(* IEC 61131-3 sources: moqui-plc/iec61131/moqui/framework/src/main/org/moqui/mqtt, 14 files *)

(* ---- MqttCmd.dut ---- *)
(*#-#-#-#-#-#-#-#-#-#---Declaration---#-#-#-#-#-#-#-#-#-#-#-#-#*)

{attribute 'qualified_only'}
{attribute 'strict'}
TYPE MqttCmd : (
	Idle := 0,
	Publish,
    Subscribe,
	Unsubscribe
); END_TYPE

(* ---- MqttCmd.st ---- *)
TYPE MqttCmd : (
	Idle := 0,
	Publish,
    Subscribe,
	Unsubscribe
); END_TYPE

(* ---- MqttConnectionRef.dut ---- *)
(*#-#-#-#-#-#-#-#-#-#---Declaration---#-#-#-#-#-#-#-#-#-#-#-#-#*)

TYPE MqttConnectionRef : STRUCT
	ref : REFERENCE TO MQTT.MQTTClient;
END_STRUCT END_TYPE

(* ---- MqttConnectionRef.st ---- *)
TYPE MqttConnectionRef : STRUCT
	ref : REFERENCE TO MQTT.MQTTClient;
END_STRUCT END_TYPE

(* ---- MqttLogAppenderStatus.dut ---- *)
(*#-#-#-#-#-#-#-#-#-#---Declaration---#-#-#-#-#-#-#-#-#-#-#-#-#*)

{attribute 'qualified_only'}
{attribute 'strict'}
TYPE MqttLogAppenderStatus : (
    Idle,
	BuildJson,
	Serialize,
	Publish,
	WaitAck
); END_TYPE

(* ---- MqttLogAppenderStatus.st ---- *)
TYPE MqttLogAppenderStatus : (
    Idle,
	BuildJson,
	Serialize,
	Publish,
	WaitAck
); END_TYPE

(* ---- MqttParameterPubStatus.dut ---- *)
(*#-#-#-#-#-#-#-#-#-#---Declaration---#-#-#-#-#-#-#-#-#-#-#-#-#*)

{attribute 'qualified_only'}
{attribute 'strict'}
TYPE MqttParameterPubStatus : (
	Idle := 0,
	BuildJson,
	Serialize,
	Publish,
	WaitAck
); END_TYPE

(* ---- MqttParameterPubStatus.st ---- *)
TYPE MqttParameterPubStatus : (
	Idle := 0,
	BuildJson,
	Serialize,
	Publish,
	WaitAck
); END_TYPE

(* ---- MqttParameterSubStatus.dut ---- *)
(*#-#-#-#-#-#-#-#-#-#---Declaration---#-#-#-#-#-#-#-#-#-#-#-#-#*)

{attribute 'qualified_only'}
{attribute 'strict'}
TYPE MqttParameterSubStatus : (
	Idle := 0,
	Subscribe,
	UpdateParameters,
	Listening,
	Error
); END_TYPE

(* ---- MqttParameterSubStatus.st ---- *)
TYPE MqttParameterSubStatus : (
	Idle := 0,
	Subscribe,
	UpdateParameters,
	Listening,
	Error
); END_TYPE

(* ---- MqttConnectionFactory.pou ---- *)
(*#-#-#-#-#-#-#-#-#-#---Declaration---#-#-#-#-#-#-#-#-#-#-#-#-#*)

{attribute 'no_assign'}
(* Component to connect with a MQTT broker, using default configurations. *)
FUNCTION_BLOCK MqttConnectionFactory
VAR_EXTERNAL CONSTANT
	brokerUrl : STRING(255);
	brokerPort : UINT;
	webSocketUrl : STRING(1024);
	clientId : STRING(255);
	username : WSTRING(255);
	password : WSTRING(1024);
	sessionExpiryInterval : UDINT;
	keepAlive : UINT;
	cleanSession : BOOL;
	timeout : UDINT;
	pingInterval : TIME;
	maximumPacketSize : UDINT;
	communicationMode : MQTT.COMMUNICATION_MODE;
	mqttVersion : MQTT.MQTT_VERSION;
	(* connectUserProperties : ARRAY [0..(MQTT.MQTTParam.g_udiMaxUserProperties - 1)] OF MQTT.MQTTStringPair; *)
	willTopic : WSTRING(1024);
	willMessage : STRING(1024);
	willRetain : BOOL;
	willQoS : MQTT.MQTT_QOS;
	willPayloadFormatIndicator : BYTE;
	willMessageExpiryInterval : UDINT;
	willContentType : WSTRING(32);
	willDelayInterval : UDINT;
END_VAR
VAR_INPUT
	connect : BOOL := TRUE;
END_VAR
VAR_OUTPUT
	connection : MQTT.MQTTClient;
    connected : BOOL;
    busy : BOOL;
    error : BOOL;
	errorId : INT;
END_VAR
VAR
	(* Connect properties v5 *)
	mqttConnectProperties : MQTT.MQTTConnectProperties := (
		udiSessionExpiryInterval := sessionExpiryInterval,
		udiMaximumPacketSize := maximumPacketSize
		(* userProperties := connectUserProperties *)
	);
	(* Will properties v5 *)
	mqttWillProperties : MQTT.MQTTWillProperties := (
		bPayloadFormatIndicator := willPayloadFormatIndicator,
		udiMessageExpiryInterval := willMessageExpiryInterval,
		wsContentType := willContentType,
		udiWillDelayInterval := willDelayInterval
		(* userProperties := willUserProperties *)
    );
	(* TLS context *)
	cipherList : NBS.CIPHER_LIST := STRUCT(psList := ADR('HIGH'), udiSize := 5);
	commonName : STRING := 'moqui';
    certInfo : NBS.CERT_INFO := (psInfo := ADR(commonName), udiSize := INT_TO_UDINT(LEN(commonName)));
	defaultTlsContext : NBS.TLSContext := (
		sUseCaseName := commonName,
		ePurpose := NBS.PURPOSE.CLIENT_SIDE,
		sTLSVersion := '1.3',
		sCipherList := cipherList,
		sHostname := brokerUrl,
		ciCertInfo := certInfo,
		udiVerificationMode	:= 2, (* 1 => No peer verification, 2 => Active Peer verification *)
		itfCertVerifer := 0
	);
	nullTlsContext : NBS.ITLSContext := 0;
	tlsContext : NBS.ITLSContext;
	useTLS : BOOL := FALSE;

	(*
     * To use client certificates, configure the connection via the TLS context.
	 * Example:
	 *      commonName : STRING := 'COMMON_NAME_OF_CERTIFICATE'; // CN of the certificate (common name).
	 *      cipherList : NBS.CIPHER_LIST := STRUCT(psList := ADR('HIGH'), udiSize := 5); // Cipher string see https://www.openssl.org/docs/man1.1.1/man1/ciphers.html
	 *      certInfo : NBS.CERT_INFO := (psInfo := ADR(commonName), udiSize := SIZEOF(commonName)); // CN of the certificate (common name)
	 *      tlsContext : NBS.TLSContext := (
	 *          sUseCaseName := commonName, // A certificate is stored in the certificate store with the use case name.
	 *          ePurpose := NBS.PURPOSE.CLIENT_SIDE, // For client certificates set this to NBS.PURPOSE.CLIENT_SIDE
     *          sTLSVersion := '1.3', // The TLS version
     *          sCipherList := cipherList, // Set the cipher list
     *          sHostname := brokerUrl, // The hostname of the broker
     *          udiVerificationMode := 2, // 2 => Active Peer verification
     *          ciCertInfo := certInfo, // Set the cert info
     *          itfCertVerifer := 0); // 0 => No Verifier
	 *      client : MQTT.MQTTClient := (itfTLSCOntext := _tlsContext);
	 * Use the method TLSContext.SetInitialValue to set the context while runtime and set the context via the input itfTLSCOntext of the client FB.
	 *)
END_VAR

(*#-#-#-#-#-#-#-#-#-#---Implementation---#-#-#-#-#-#-#-#-#-#-#-#-#*)

(* TLS selection *)
tlsContext := nullTlsContext;
IF useTLS THEN tlsContext := defaultTlsContext; END_IF;

(* Configure the MQTT connection *)
connection(xEnable := connect, xConnectedToBroker => connected, xError => error, eMQTTerror => errorId,
	sHostname := brokerUrl, uiPort := brokerPort, sWebSocketUrl := webSocketUrl, sClientId := clientId,
	itfTLSContext := tlsContext, eCommunicationMode := communicationMode, eMQTTVersion := mqttVersion,
	wsUsername := username, wsPassword := password, mQTTConnectProperties := mqttConnectProperties,
	uiKeepAlive := keepAlive, xCleanSession := cleanSession, udiTimeOut := timeout, tPingInterval := pingInterval,
	wsWillTopic := willTopic, pbWillMessage := ADR(willMessage), uiWillMessageSize := INT_TO_UINT(LEN(willMessage)),
	xWillRetain := willRetain, eWillQoS := willQoS, mQTTWillProperties := mqttWillProperties);

(* ---- MqttConnectionFactory.st ---- *)
(* Component to connect with a MQTT broker, using default configurations. *)
FUNCTION_BLOCK MqttConnectionFactory
	VAR_EXTERNAL CONSTANT
		brokerUrl : STRING(255);
		brokerPort : UINT;
		webSocketUrl : STRING(1024);
		clientId : STRING(255);
		username : WSTRING(255);
		password : WSTRING(1024);
		sessionExpiryInterval : UDINT;
		keepAlive : UINT;
		cleanSession : BOOL;
		timeout : UDINT;
		pingInterval : TIME;
		maximumPacketSize : UDINT;
		communicationMode : MQTT.COMMUNICATION_MODE;
		mqttVersion : MQTT.MQTT_VERSION;
		(* connectUserProperties : ARRAY [0..(MQTT.MQTTParam.g_udiMaxUserProperties - 1)] OF MQTT.MQTTStringPair; *)
		willTopic : WSTRING(1024);
		willMessage : STRING(1024);
		willRetain : BOOL;
		willQoS : MQTT.MQTT_QOS;
		willPayloadFormatIndicator : BYTE;
		willMessageExpiryInterval : UDINT;
		willContentType : WSTRING(32);
		willDelayInterval : UDINT;
	END_VAR
	VAR_INPUT
		connect : BOOL := TRUE;
	END_VAR
	VAR_OUTPUT
		connection : MQTT.MQTTClient;
	    connected : BOOL;
	    busy : BOOL;
	    error : BOOL;
		errorId : INT;
	END_VAR
	VAR
		(* Connect properties v5 *)
		mqttConnectProperties : MQTT.MQTTConnectProperties := (
			udiSessionExpiryInterval := sessionExpiryInterval,
			udiMaximumPacketSize := maximumPacketSize
			(* userProperties := connectUserProperties *)
		);
		(* Will properties v5 *)
		mqttWillProperties : MQTT.MQTTWillProperties := (
			bPayloadFormatIndicator := willPayloadFormatIndicator,
			udiMessageExpiryInterval := willMessageExpiryInterval,
			wsContentType := willContentType,
			udiWillDelayInterval := willDelayInterval
			(* userProperties := willUserProperties *)
	    );
		(* TLS context *)
		cipherList : NBS.CIPHER_LIST := STRUCT(psList := ADR('HIGH'), udiSize := 5);
		commonName : STRING := 'moqui';
	    certInfo : NBS.CERT_INFO := (psInfo := ADR(commonName), udiSize := INT_TO_UDINT(LEN(commonName)));
		defaultTlsContext : NBS.TLSContext := (
			sUseCaseName := commonName,
			ePurpose := NBS.PURPOSE.CLIENT_SIDE,
			sTLSVersion := '1.3',
			sCipherList := cipherList,
			sHostname := brokerUrl,
			ciCertInfo := certInfo,
			udiVerificationMode	:= 2, (* 1 => No peer verification, 2 => Active Peer verification *)
			itfCertVerifer := 0
		);
		nullTlsContext : NBS.ITLSContext := 0;
		tlsContext : NBS.ITLSContext;
		useTLS : BOOL := FALSE;

		(*
	     * To use client certificates, configure the connection via the TLS context.
		 * Example:
		 *      commonName : STRING := 'COMMON_NAME_OF_CERTIFICATE'; // CN of the certificate (common name).
		 *      cipherList : NBS.CIPHER_LIST := STRUCT(psList := ADR('HIGH'), udiSize := 5); // Cipher string see https://www.openssl.org/docs/man1.1.1/man1/ciphers.html
		 *      certInfo : NBS.CERT_INFO := (psInfo := ADR(commonName), udiSize := SIZEOF(commonName)); // CN of the certificate (common name)
		 *      tlsContext : NBS.TLSContext := (
		 *          sUseCaseName := commonName, // A certificate is stored in the certificate store with the use case name.
		 *          ePurpose := NBS.PURPOSE.CLIENT_SIDE, // For client certificates set this to NBS.PURPOSE.CLIENT_SIDE
	     *          sTLSVersion := '1.3', // The TLS version
	     *          sCipherList := cipherList, // Set the cipher list
	     *          sHostname := brokerUrl, // The hostname of the broker
	     *          udiVerificationMode := 2, // 2 => Active Peer verification
	     *          ciCertInfo := certInfo, // Set the cert info
	     *          itfCertVerifer := 0); // 0 => No Verifier
		 *      client : MQTT.MQTTClient := (itfTLSCOntext := _tlsContext);
		 * Use the method TLSContext.SetInitialValue to set the context while runtime and set the context via the input itfTLSCOntext of the client FB.
		 *)
	END_VAR

	(* TLS selection *)
	tlsContext := nullTlsContext;
	IF useTLS THEN tlsContext := defaultTlsContext; END_IF;

	(* Configure the MQTT connection *)
	connection(xEnable := connect, xConnectedToBroker => connected, xError => error, eMQTTerror => errorId,
		sHostname := brokerUrl, uiPort := brokerPort, sWebSocketUrl := webSocketUrl, sClientId := clientId,
		itfTLSContext := tlsContext, eCommunicationMode := communicationMode, eMQTTVersion := mqttVersion,
		wsUsername := username, wsPassword := password, mQTTConnectProperties := mqttConnectProperties,
		uiKeepAlive := keepAlive, xCleanSession := cleanSession, udiTimeOut := timeout, tPingInterval := pingInterval,
		wsWillTopic := willTopic, pbWillMessage := ADR(willMessage), uiWillMessageSize := INT_TO_UINT(LEN(willMessage)),
		xWillRetain := willRetain, eWillQoS := willQoS, mQTTWillProperties := mqttWillProperties);
	END_FUNCTION_BLOCK

(* ---- MqttLogAppender.pou ---- *)
(*#-#-#-#-#-#-#-#-#-#---Declaration---#-#-#-#-#-#-#-#-#-#-#-#-#*)

{attribute 'no_assign'}
FUNCTION_BLOCK MqttLogAppender
VAR_EXTERNAL CONSTANT
    LOG_MAX_SIZE : UINT;
	LOG_JSON_PAYLOAD_MAX_SIZE : UINT;
	pubPayloadFormatIndicator : BYTE;
	pubMessageExpiryInterval : UDINT;
	pubContentType : WSTRING(32);
	(* pubUserProperties : ARRAY [0..(MQTT.MQTTParam.g_udiMaxUserProperties - 1)] OF MQTT.MQTTStringPair; *)
	logPubQoS : MQTT.MQTT_QOS;
	logPubRetain : BOOL;
	logReDelivery : BOOL;
	logTopic : WSTRING(1024);
	logAppenderTimeout : UINT;
END_VAR
VAR_EXTERNAL
	connectionFactory : MqttConnectionFactory;
END_VAR
VAR_INPUT
    execute : BOOL;
    (* Data sources *)
    logBuffer : REFERENCE TO ARRAY[1..LOG_MAX_SIZE] OF LogEvent;
    logBufferSize : UINT;
END_VAR
VAR_OUTPUT
	done, busy, error : BOOL;
    errorId : INT; (* 100 : ArgsErr *)
END_VAR
VAR
	pubTopic : WSTRING(1024) := logTopic;
	(* Publisher *)
	publisher : MQTT.MQTTPublish;
	(* Publish properties v5 *)
	mqttPublishProperties : MQTT.MQTTPublishProperties := (
		bPayloadFormatIndicator := pubPayloadFormatIndicator,
		wsContentType := pubContentType,
		udiMessageExpiryInterval := pubMessageExpiryInterval
		(* userProperties := pubUserProperties *)
	);
    (* JSON serializer *)
    logMapper : SerializeLogToJson;
END_VAR

(*#-#-#-#-#-#-#-#-#-#---Implementation---#-#-#-#-#-#-#-#-#-#-#-#-#*)

IF NOT execute THEN
	logMapper(execute := FALSE, done => done, busy => busy,
		error => error, errorId => errorId);
    publisher(xExecute := FALSE, mqttClient := connectionFactory.connection, wsTopicName := pubTopic,
		xDone => done, xBusy => busy, xError => error, eMQTTError => errorId);
	RETURN;
END_IF;

(* Connect to the broker *)
connectionFactory(connect := TRUE, error => error, errorId => errorId);
(* Reset and retry on next cycle *)
IF connectionFactory.error THEN
	connectionFactory(connect := FALSE, error => error, errorId => errorId);
	done := FALSE; busy := FALSE;
	RETURN;
END_IF;

(* Waiting for connection to broker *)
IF NOT connectionFactory.connected THEN RETURN; END_IF;

IF NOT publisher.xBusy THEN
	(* JSON mapping *)
	logMapper(execute := TRUE, logBuffer := logBuffer, logBufferSize := logBufferSize,
		lineBreak := "", (* compact output: avoid WSTRING line-break embedding null bytes in byte array *)
		busy => busy, error => error, errorId => errorId);
	IF logMapper.error THEN
		(* Reset JSON writer *)
		logMapper(execute := FALSE, busy => busy,
			error => error, errorId => errorId);
		done := FALSE; busy := FALSE;
		RETURN;
	END_IF;
END_IF;

IF logMapper.done THEN
	(* Publish the payload *)
	publisher(xExecute := TRUE, mqttClient := connectionFactory.connection, wsTopicName := pubTopic,
		pbPayload := ADR(logMapper.jsonPayload), udiPayloadSize := logMapper.payloadSize,
		eQoS := logPubQoS, xReDelivery := logReDelivery, xRetain := logPubRetain,
		udiTimeOut := UINT_TO_UDINT(logAppenderTimeout), mQTTPublishProperties := mqttPublishProperties,
		xDone => done, xBusy => busy, xError => error, eMQTTError => errorId);
END_IF;

(* ---- MqttLogAppender.st ---- *)
FUNCTION_BLOCK MqttLogAppender
	VAR_EXTERNAL CONSTANT
	    LOG_MAX_SIZE : UINT;
		LOG_JSON_PAYLOAD_MAX_SIZE : UINT;
		pubPayloadFormatIndicator : BYTE;
		pubMessageExpiryInterval : UDINT;
		pubContentType : WSTRING(32);
		(* pubUserProperties : ARRAY [0..(MQTT.MQTTParam.g_udiMaxUserProperties - 1)] OF MQTT.MQTTStringPair; *)
		logPubQoS : MQTT.MQTT_QOS;
		logPubRetain : BOOL;
		logReDelivery : BOOL;
		logTopic : WSTRING(1024);
		logAppenderTimeout : UINT;
	END_VAR
	VAR_EXTERNAL
		connectionFactory : MqttConnectionFactory;
	END_VAR
	VAR_INPUT
	    execute : BOOL;
	    (* Data sources *)
	    logBuffer : REFERENCE TO ARRAY[1..LOG_MAX_SIZE] OF LogEvent;
	    logBufferSize : UINT;
	END_VAR
	VAR_OUTPUT
		done, busy, error : BOOL;
	    errorId : INT; (* 100 : ArgsErr *)
	END_VAR
	VAR
		pubTopic : WSTRING(1024) := logTopic;
		(* Publisher *)
		publisher : MQTT.MQTTPublish;
		(* Publish properties v5 *)
		mqttPublishProperties : MQTT.MQTTPublishProperties := (
			bPayloadFormatIndicator := pubPayloadFormatIndicator,
			wsContentType := pubContentType,
			udiMessageExpiryInterval := pubMessageExpiryInterval
			(* userProperties := pubUserProperties *)
		);
	    (* JSON serializer *)
	    logMapper : SerializeLogToJson;
	END_VAR

	IF NOT execute THEN
		logMapper(execute := FALSE, done => done, busy => busy,
			error => error, errorId => errorId);
	    publisher(xExecute := FALSE, mqttClient := connectionFactory.connection, wsTopicName := pubTopic,
			xDone => done, xBusy => busy, xError => error, eMQTTError => errorId);
		RETURN;
	END_IF;

	(* Connect to the broker *)
	connectionFactory(connect := TRUE, error => error, errorId => errorId);
	(* Reset and retry on next cycle *)
	IF connectionFactory.error THEN
		connectionFactory(connect := FALSE, error => error, errorId => errorId);
		done := FALSE; busy := FALSE;
		RETURN;
	END_IF;

	(* Waiting for connection to broker *)
	IF NOT connectionFactory.connected THEN RETURN; END_IF;

	IF NOT publisher.xBusy THEN
		(* JSON mapping *)
		logMapper(execute := TRUE, logBuffer := logBuffer, logBufferSize := logBufferSize,
			lineBreak := "", (* compact output: avoid WSTRING line-break embedding null bytes in byte array *)
			busy => busy, error => error, errorId => errorId);
		IF logMapper.error THEN
			(* Reset JSON writer *)
			logMapper(execute := FALSE, busy => busy,
				error => error, errorId => errorId);
			done := FALSE; busy := FALSE;
			RETURN;
		END_IF;
	END_IF;

	IF logMapper.done THEN
		(* Publish the payload *)
		publisher(xExecute := TRUE, mqttClient := connectionFactory.connection, wsTopicName := pubTopic,
			pbPayload := ADR(logMapper.jsonPayload), udiPayloadSize := logMapper.payloadSize,
			eQoS := logPubQoS, xReDelivery := logReDelivery, xRetain := logPubRetain,
			udiTimeOut := UINT_TO_UDINT(logAppenderTimeout), mQTTPublishProperties := mqttPublishProperties,
			xDone => done, xBusy => busy, xError => error, eMQTTError => errorId);
	END_IF;
	END_FUNCTION_BLOCK
